TYPE ST_MPC_Matrices :
STRUCT
	gMPC_F : ARRAY[1..20,1..2] OF LREAL := [-10.110286651796301,-0.494890603179854,
											-9.998121030930005,-0.849211680989655,
											-9.882750302704293,-1.186962702093454,
											-9.764412993557139,-1.508607889096049,
											-9.643339387385019,-1.814603927230396,
											-9.519751705206597,-2.105399926086415,
											-9.393864283415191,-2.381437389289509,
											-9.265883750536544,-2.643150191797635,
											-9.136009202413343,-2.890964564494386,
											-9.004432375742766,-3.125299085763932,
											-8.871337819898013,-3.346564679742028,
											-8.736903066969232,-3.555164620945482,
											-8.601298799963665,-3.751494544990575,
											-8.464689019109006,-3.935942465118846,
											-8.327231206208078,-4.108888794256542,
											-8.189076486996795,-4.270706372341670,
											-8.050369791461257,-4.421760498660247,
											-7.911250012073411,-4.562408968940717,
											-7.771850159908285,-4.693002116962906,
											-7.632297518609167,-4.813882860445012];

	gMPC_Phi : ARRAY[1..20,1..5] OF LREAL := [0.000284731809204,0.000000000000000,0.000000000000000,0.000000000000000,0.000000000000000,
											0.000363650992320,0.000284731809204,0.000000000000000,0.000000000000000,0.000000000000000,
											0.000438735836864,0.000363650992320,0.000284731809204,0.000000000000000,0.000000000000000,
											0.000510096292665,0.000438735836864,0.000363650992320,0.000284731809204,0.000000000000000,
											0.000577840450081,0.000510096292665,0.000438735836864,0.000363650992320,0.000284731809204,
											0.000642074534315,0.000577840450081,0.000510096292665,0.000438735836864,0.000363650992320,
											0.000702902901532,0.000642074534315,0.000577840450081,0.000510096292665,0.000438735836864,
											0.000760428036683,0.000702902901532,0.000642074534315,0.000577840450081,0.000510096292665,
											0.000814750552970,0.000760428036683,0.000702902901532,0.000642074534315,0.000577840450081,
											0.000865969192870,0.000814750552970,0.000760428036683,0.000702902901532,0.000642074534315,
											0.000914180830659,0.000865969192870,0.000814750552970,0.000760428036683,0.000702902901532,
											0.000959480476359,0.000914180830659,0.000865969192870,0.000814750552970,0.000760428036683,
											0.001001961281039,0.000959480476359,0.000914180830659,0.000865969192870,0.000814750552970,
											0.001041714543414,0.001001961281039,0.000959480476359,0.000914180830659,0.000865969192870,
											0.001078829717667,0.001041714543414,0.001001961281039,0.000959480476359,0.000914180830659,
											0.001113394422447,0.001078829717667,0.001041714543414,0.001001961281039,0.000959480476359,
											0.001145494450968,0.001113394422447,0.001078829717667,0.001041714543414,0.001001961281039,
											0.001175213782158,0.001145494450968,0.001113394422447,0.001078829717667,0.001041714543414,
											0.001202634592808,0.001175213782158,0.001145494450968,0.001113394422447,0.001078829717667,
											0.001227837270652,0.001202634592808,0.001175213782158,0.001145494450968,0.001113394422447];

	gMPC_H : ARRAY[1..5,1..5] OF LREAL := [0.100015794350270,0.000014974076270,0.000014113898875,0.000013221055499,0.000012302759971,
											0.000014974076270,0.100014286765906,0.000013497436694,0.000012670927592,0.000011814574719,
											0.000014113898875,0.000013497436694,0.100012840435943,0.000012084083946,0.000011293316339,
											0.000013221055499,0.000012670927592,0.000012084083946,0.100011459308509,0.000010737883080,
											0.000012302759971,0.000011814574719,0.000011293316339,0.000010737883080,0.100010147150972];

	gMPC_Hinv : ARRAY[1..5,1..5] OF LREAL := [9.998421563375079,-0.001496454423596,-0.001410485502700,-0.001321253378510,-0.001229479083734,
												-0.001496454423596,9.998572233479088,-0.001348880189337,-0.001266279112390,-0.001180696570227,
												-0.001410485502700,-0.001348880189337,9.998716775705333,-0.001207636356411,-0.001128609625938,
												-0.001321253378510,-0.001266279112390,-0.001207636356411,9.998854796675317,-0.001073107909165,
												-0.001229479083734,-0.001180696570227,-0.001128609625938,-0.001073107909165,9.998985921243611];
END_STRUCT
END_TYPE

(* stored: Version 1.1.0.1, ProductVersion 3.1.4024.9
   DUT ST_MPC_Matrices: Id {a8a01b78-9e78-4520-8161-00057664ce98} *)
